FUNCTION_BLOCK FB_SwitchHoming IMPLEMENTS I_MotionSequence
VAR_INPUT
	HomingParameter	: MC_HomingParameter;
END_VAR
VAR_OUTPUT
	State	: UINT;
END_VAR
VAR
	diHomeSwitch	AT %I* : BOOL;
	doHomeSwitch	AT %Q* : BOOL := TRUE;
	validaxisref	: BOOL := FALSE;
	_Axis			: SPT_Motion_Control.I_BasicAxis;
	Home			: MC_Home;
END_VAR

{warning 'Add property implementation'}
PROPERTY Axis : SPT_Motion_Control.I_BasicAxis
GET
Axis	:= _Axis;
END_GET
SET
_Axis	:= Axis;
validaxisref	:= TRUE;
END_SET
END_PROPERTY

{warning 'Add property implementation'}
PROPERTY Busy : BOOL
GET
END_GET
END_PROPERTY

{warning 'Add method implementation '}
METHOD CyclicLogic
IF validaxisref THEN
	Home.bCalibrationCam	:= diHomeSwitch;
	Home(Axis := _Axis.Axis);

END_IF

IF NOT Home.Execute	THEN
	State	:= 0;
END_IF
Home.Execute	:= FALSE;
END_METHOD

{warning 'Add property implementation'}
PROPERTY Error : BOOL
GET
END_GET
END_PROPERTY

{warning 'Add property implementation'}
PROPERTY ErrorID : UDINT
GET
END_GET
END_PROPERTY

{warning 'Add method implementation '}
METHOD Execute : BOOL
Home.Execute					:= TRUE;
Home.Position					:= 39;
Home.HomingMode					:= MC_DefaultHoming;
Home.Options.SearchVelocity		:= 50;
Home.Options.SearchDirection	:= MC_Negative_Direction;

// return true when done
Execute	:= Home.Done;
END_METHOD

{warning 'Add property implementation'}
PROPERTY InitComplete : BOOL
GET
END_GET
END_PROPERTY

END_FUNCTION_BLOCK

(* stored: Version 1.1.0.1
   POU FB_SwitchHoming: Id {6cba173b-6846-48ee-9db1-475d58063724}, SpecialFunc None
   Property Axis: Id {a3a1b938-cb76-468b-986b-717edf4e6395}
   Get Get: Id {d0c686b8-36c9-4819-99c3-bc060ce836d4}
   Set Set: Id {d321e3e3-5950-4d70-ba9a-a5c1172b9dd4}
   Property Busy: Id {019f1f96-8c2b-4fe6-94c4-92fc90967329}
   Get Get: Id {1312500b-8109-485b-9bec-228604416438}
   Method CyclicLogic: Id {8eb2b983-7c4a-41b5-9333-dc0e7dfec0a3}
   Property Error: Id {ac6eaf90-008b-4873-b53b-df509f1d654c}
   Get Get: Id {dcad8511-7533-46ac-87e5-607cfb2d9194}
   Property ErrorID: Id {abd6fe9d-9a72-4974-8125-4aba519d27be}
   Get Get: Id {c1289d1e-9738-49aa-af94-7c8be41b2db6}
   Method Execute: Id {5cc5614b-803d-45d5-b1f5-18dc23f621b1}
   Property InitComplete: Id {636bfefc-5a41-493e-9693-11a02231145e}
   Get Get: Id {031192f9-9823-4747-9e4d-9adf5bd436d8} *)
